{attribute 'pack_mode' := '2'}
TYPE ST_XTS_TRANSPORT_CTRL :
STRUCT
  Cmd       : E_XTS_TRANSPORT_CTRL;
END_STRUCT
END_TYPE

(* stored: Version 1.1.0.1, ProductVersion 3.1.4026.18
   DUT ST_XTS_TRANSPORT_CTRL: Id {b339479e-6cb2-4ce2-a1e3-95a809318168} *)
